Universal Robots PolyScope program: Dance.urp

Program Dance (installation=default directory=/programs createdIn=5.12.5.10626004 lastSavedIn=5.12.5.10626004 robotSerialNumber=)
Robot Program (runOnlyOnce=false)
  'Multi-stage dance: wake / bow / sweep / surge / wave / spiral / flourish / home'
  Script file /programs/dance.script
    | def dance():
    |   textmsg("dance/stage=wake")
    |   movej([-0.7427, -1.9034, -2.1358, -0.3718, 1.5714, 2.3782], a=0.8, v=0.6, r=0.05)
    |   textmsg("dance/stage=bow")
    |   movej([-0.7427, -2.4034, -2.7358, 0.4282, 1.5714, 2.3782], a=0.8, v=0.5)
    |   sleep(0.4)
    |   movej([-0.7427, -1.9034, -2.1358, -0.3718, 1.5714, 2.3782], a=1.0, v=0.8, r=0.05)
    |   textmsg("dance/stage=sweep")
    |   movej([0.0573, -2.0034, -2.2358, -0.2718, 1.5714, 1.9782], a=1.2, v=1.0, r=0.08)
    |   movej([-1.5427, -2.0034, -2.2358, -0.2718, 1.5714, 2.7782], a=1.2, v=1.0, r=0.08)
    |   movej([0.0573, -2.0034, -2.2358, -0.2718, 1.5714, 1.9782], a=1.2, v=1.0, r=0.08)
    |   movej([-1.5427, -2.0034, -2.2358, -0.2718, 1.5714, 2.7782], a=1.2, v=1.0, r=0.08)
    |   movej([-0.7427, -1.9034, -2.1358, -0.3718, 1.5714, 2.3782], a=1.2, v=0.9, r=0.05)
    |   textmsg("dance/stage=surge")
    |   movej([-0.7427, -1.7534, -1.9358, -0.5718, 1.5714, 2.3782], a=1.6, v=1.3, r=0.04)
    |   movej([-0.7427, -2.3534, -2.7358, 0.2282, 1.5714, 2.3782], a=1.6, v=1.3, r=0.04)
    |   movej([-0.7427, -1.7534, -1.9358, -0.5718, 1.5714, 2.3782], a=1.6, v=1.3, r=0.04)
    |   movej([-0.7427, -2.3534, -2.7358, 0.2282, 1.5714, 2.3782], a=1.6, v=1.3, r=0.04)
    |   movej([-0.7427, -1.7534, -1.9358, -0.5718, 1.5714, 2.3782], a=1.6, v=1.3, r=0.04)
    |   movej([-0.7427, -2.3534, -2.7358, 0.2282, 1.5714, 2.3782], a=1.6, v=1.3, r=0.04)
    |   movej([-0.7427, -1.9034, -2.1358, -0.3718, 1.5714, 2.3782], a=1.2, v=0.9, r=0.05)
    |   textmsg("dance/stage=wave")
    |   movej([-0.5427, -2.0034, -2.3358, -0.4718, 1.7714, 3.1782], a=1.5, v=1.2, r=0.05)
    |   movej([-0.5427, -2.0034, -2.3358, 0.3282, 1.3714, 1.5782], a=1.5, v=1.2, r=0.05)
    |   movej([-0.9427, -2.0034, -2.3358, -0.4718, 1.7714, 3.1782], a=1.5, v=1.2, r=0.05)
    |   movej([-0.9427, -2.0034, -2.3358, 0.3282, 1.3714, 1.5782], a=1.5, v=1.2, r=0.05)
    |   movej([-0.5427, -2.0034, -2.3358, -0.4718, 1.7714, 3.1782], a=1.5, v=1.2, r=0.05)
    |   movej([-0.5427, -2.0034, -2.3358, 0.3282, 1.3714, 1.5782], a=1.5, v=1.2, r=0.05)
    |   movej([-0.7427, -1.9034, -2.1358, -0.3718, 1.5714, 2.3782], a=1.2, v=0.9, r=0.05)
    |   textmsg("dance/stage=spiral")
    |   movej([-0.7427, -1.7034, -2.1358, -0.4718, 1.5714, -0.6218], a=1.4, v=1.4, r=0.06)
    |   movej([-0.7427, -1.7034, -2.1358, -0.4718, 1.5714, 0.8782], a=1.4, v=1.4, r=0.06)
    |   movej([-0.7427, -1.7034, -2.1358, -0.4718, 1.5714, 2.3782], a=1.4, v=1.4, r=0.06)
    |   movej([-0.7427, -1.7034, -2.1358, -0.4718, 1.5714, 3.8782], a=1.4, v=1.4, r=0.06)
    |   movej([-0.7427, -1.7034, -2.1358, -0.4718, 1.5714, 5.3782], a=1.4, v=1.4, r=0.06)
    |   movej([-0.7427, -1.7034, -2.1358, -0.4718, 1.5714, 3.8782], a=1.4, v=1.4, r=0.06)
    |   movej([-0.7427, -1.7034, -2.1358, -0.4718, 1.5714, 2.3782], a=1.4, v=1.4, r=0.06)
    |   movej([-0.7427, -1.7034, -2.1358, -0.4718, 1.5714, 0.8782], a=1.4, v=1.4)
    |   textmsg("dance/stage=flourish")
    |   movej([-0.2427, -1.9034, -2.2358, -0.3718, 1.5714, 1.1782], a=1.6, v=1.3, r=0.06)
    |   movej([-1.2427, -1.9034, -2.2358, -0.3718, 1.5714, 3.5782], a=1.6, v=1.3, r=0.06)
    |   movej([-0.2427, -1.9034, -2.2358, -0.3718, 1.5714, 1.1782], a=1.6, v=1.3, r=0.06)
    |   textmsg("dance/stage=home")
    |   movej([-0.7427, -2.1034, -2.5358, -0.0718, 1.5714, 2.3782], a=0.8, v=0.6)
    |   sleep(0.8)
    |   sync()
    | end
  Script: dance()
